// TIA Portal V20 export
TYPE "typeCmControlNodeSoftCamtransferPnPRightAxisY"
// stored: Namespace Unit1.Em5
   STRUCT
      pos00_wait : "LER_typeSoftCamPosition";
      pos01_hipotThickness : "LER_typeSoftCamPosition";
      pos02_vision : "LER_typeSoftCamPosition";
      pos03_laserMark : "LER_typeSoftCamPosition";
      pos04_weightCheck : "LER_typeSoftCamPosition";
      pos05_position : "LER_typeSoftCamPosition";
      pos06_position : "LER_typeSoftCamPosition";
      pos07_position : "LER_typeSoftCamPosition";
      pos08_noInterferenceZone : "LER_typeSoftCamPosition";
      pos09_position : "LER_typeSoftCamPosition";
      pos10_position : "LER_typeSoftCamPosition";
      pos11_position : "LER_typeSoftCamPosition";
      pos12_position : "LER_typeSoftCamPosition";
      pos13_position : "LER_typeSoftCamPosition";
      pos14_position : "LER_typeSoftCamPosition";
      pos15_position : "LER_typeSoftCamPosition";
   END_STRUCT;
END_TYPE
